// TIA Portal V19 export
DATA_BLOCK "DB_PointerHMI"   // DB25
{ S7_Optimized_Access := 'TRUE'; DB_Accessible_From_OPC_UA := 'FALSE' }
// stored: AutoNumber false, DBAccessibleFromOPCUA false, DBAccessibleFromWebserver false, MemoryReserve 100
   VAR
      Coordination : Word;
      ProjectID : Word;
      ScreenNumber : Array[0..4] of Word;
      JobMailbox : Array[0..3] of Word;
   END_VAR
BEGIN
END_DATA_BLOCK
